TYPE ST_Param :
STRUCT
	stStatus:ST_ParamStatus;	//informations d'états (compteur de pièces, modes,...)
	stFixed:ST_ParamFixed;		//Paramètres pas en lien avec le produit, fixe
	stRecipe:ST_ParamRecipe;	//Paramètres en lien avec le produit
	stMachine:ST_ParamMachine;	//Parametres de la machine
END_STRUCT
END_TYPE

(* stored: Version 1.1.0.1, ProductVersion 3.1.4020.12
   DUT ST_Param: Id {2a98fcc6-f014-4526-94c4-e84e06f6fba5} *)
